// TIA Portal V18 export
TYPE "UDT_MES_LoadDatae_ext"
// stored: IsFailsafeCompliant false
   STRUCT
      "PLC.PartTypeID" : Int;   // 产品类型
      "PLC.PartSN" : String[50];   // 产品主体码
      "PLC.SubPartID" : String[50];   // 产品组件码
      "MES.ErrorCode" : Int;   // 异常代码
      "MES.ErrorMsg" : String[50];   // 异常信息
      "MES.StatusBits" : DInt;   // 产品状态
      "MES.Cycle_ID" : DInt;
      "MES.Unit_ParttypeID" : Int;
   END_STRUCT;
END_TYPE
